// TIA Portal project "HandlingDevice" (V13)

(* hardware
DEVICE "S7300/ET200M-Station_1"  S7-300 station
   slot 0: "Profilschiene_0"  Rail  6ES7 390-1***0-0AA0
   slot 1: "PS 307 2A_1"  PS 307 2A  6ES7 307-1BA00-0AA0
   slot 2: "PLC_1"  CPU 314C-2 PN/DP  6ES7 314-6EH04-0AB0  V3.3
      slot 2: "PROFINET-Schnittstelle_1"  PN-IO
         slot 1: "Port_1"  Port
         slot 2: "Port_2"  Port
      slot 5: "DI 24/DO 16_1"  DI24/DO16
      slot 6: "AI 5/AO 2_1"  AI5/AO2
      slot 7: "Zählen_1"  Counter
      slot 8: "Positionieren_1"  Positioning
*)

// ===== PLC "PLC_1"  CPU 314C-2 PN/DP =====

VAR_GLOBAL   // PLC tag table "Standard-Variablentabelle"
   "1S1" AT %I124.0 : Bool;   // Start-Taster (NO)
   "2S1" AT %E124.1 : Bool;   // Halt-Taster (NC)
   "3S1" AT %E124.2 : Bool;   // Richten-Taster (NO)
   "1B1" AT %E124.3 : Bool;   // Zylinder A eingefahren
   "1B2" AT %E124.4 : Bool;   // Zylinder A ausgefahren
   "2B1" AT %E124.5 : Bool;   // Zylinder C in Position unten (eingefahren)
   "2B2" AT %E124.6 : Bool;   // Zylinder C in Position Werkstückaufnahme/-übergabe
   "3B1" AT %E124.7 : Bool;   // Drehtisch D in Position Werkstückaufnahme
   "3B2" AT %E125.0 : Bool;   // Drehtisch D in Position Werkstückübergabe
   "4B1" AT %E125.1 : Bool;   // Schlitten E in Position oben
   "4B2" AT %E125.2 : Bool;   // Schlitten E in Position Werkstückaufnahme/-übergabe
   "5B1" AT %E125.3 : Bool;   // Drehantrieb F in Position Werkstückaufnahme
   "5B2" AT %E125.4 : Bool;   // Drehantrieb F in Position Werkstückübergabe
   "6B1" AT %E125.5 : Bool;   // Werkstück am Greifer A angesaugt
   "6B2" AT %E125.6 : Bool;   // Werkstück am Greifer F angesaugt
   "1M1" AT %A124.0 : Bool;   // Zylinder A ausfahren
   "2M1" AT %A124.1 : Bool;   // Drehantrieb A in Position Werkstückaufnahme drehen
   "2M2" AT %A124.2 : Bool;   // Drehantrieb A in Position Werkstückübergabe drehen
   "3M1" AT %A124.3 : Bool;   // Zylinder C in Position Werkstückaufnahme/-übergabe
   "4M1" AT %A124.4 : Bool;   // Drehtisch D in Position Werkstückübergabe drehen
   "4M2" AT %A124.5 : Bool;   // Drehtisch D in Position Werkstückaufnahme drehen
   "5M1" AT %A124.6 : Bool;   // Schlitten E in Position Werkstückaufnahme/-übergabe fahren
   "6M1" AT %A124.7 : Bool;   // Drehantrieb F in Position Werkstückübergabe drehen
   "6M2" AT %A125.0 : Bool;   // Drehantrieb F in Position Werkstückaufnahme drehen
   "7M1" AT %A125.1 : Bool;   // Vakuum Greifer A einschalten
   "7M2" AT %A125.2 : Bool;   // Vakuum Greifer A ausschalten
   "8M1" AT %A125.3 : Bool;   // Vakuum Greifer F einschalten
   "8M2" AT %A125.4 : Bool;   // Vakuum Greifer F ausschalten
   "P_S" AT %A125.5 : Bool;   // Startlampe (grün)
   "P_H" AT %A125.6 : Bool;   // Haltlampe (rot)
   "P_R" AT %A125.7 : Bool;   // Richtenlampe (orange)
   "Step0" AT %M0.0 : Bool;   // Step0
   "Step1" AT %M0.1 : Bool;   // Step1
   "Step2" AT %M0.2 : Bool;   // Step2
   "Step3" AT %M0.3 : Bool;   // Step3
   "Step4" AT %M0.4 : Bool;   // Step4
   "Step5" AT %M0.5 : Bool;   // Step5
   "Step5.1" AT %M10.0 : Bool;   // Step5.1
   "Step5.2" AT %M10.1 : Bool;   // Step5.2
   "Step5.3" AT %M10.2 : Bool;   // Step5.3
   "Step5.4" AT %M10.3 : Bool;   // Step5.4
   "Step5.5" AT %M10.4 : Bool;   // Step5.5
   "Step5.6" AT %M10.5 : Bool;   // Step5.6
   "Step5.7" AT %M10.6 : Bool;   // Step5.7
   "Step5.8" AT %M10.7 : Bool;   // Step5.8
   "Step5.9" AT %M11.0 : Bool;   // Step5.9
   "Step5.10" AT %M11.1 : Bool;   // Step5.10
   "Step5.11" AT %M11.2 : Bool;   // Step5.11
   "Step5.12" AT %M11.3 : Bool;   // Step5.12
   "Step5.13" AT %M11.4 : Bool;   // Step5.13
   "Step5.14" AT %M11.5 : Bool;   // Step5.14
   "Step5.15" AT %M11.6 : Bool;   // Step5.15
   "Step5.16" AT %M11.7 : Bool;   // Step5.16
   "Step5.17" AT %M12.0 : Bool;   // Step5.17
   "InitialStep" AT %M20.0 : Bool;   // Intiral Step
   "Mx_Gerichtet" AT %M1.0 : Bool;   // Anlage Gerichtet
   "Mx_Ausgangstellung" AT %M1.1 : Bool;   // Anlage in Ausgangstellung
   "Mx_Start" AT %M1.2 : Bool;
   "Tag_1" AT %MW0 : Int;
   "Tag_2" AT %MD10 : DWord;
   "Tag_3" AT %M1.3 : Bool;
   "Tag_4" AT %QW124 : Word;
   "Tag_5" AT %M1.4 : Bool;
END_VAR

FUNCTION "FC1 Grafcet G1" : Void   // FC1, FBD
{ S7_Optimized_Access := 'FALSE' }
VERSION : 0.1
BEGIN

REGION Network 1: Step0
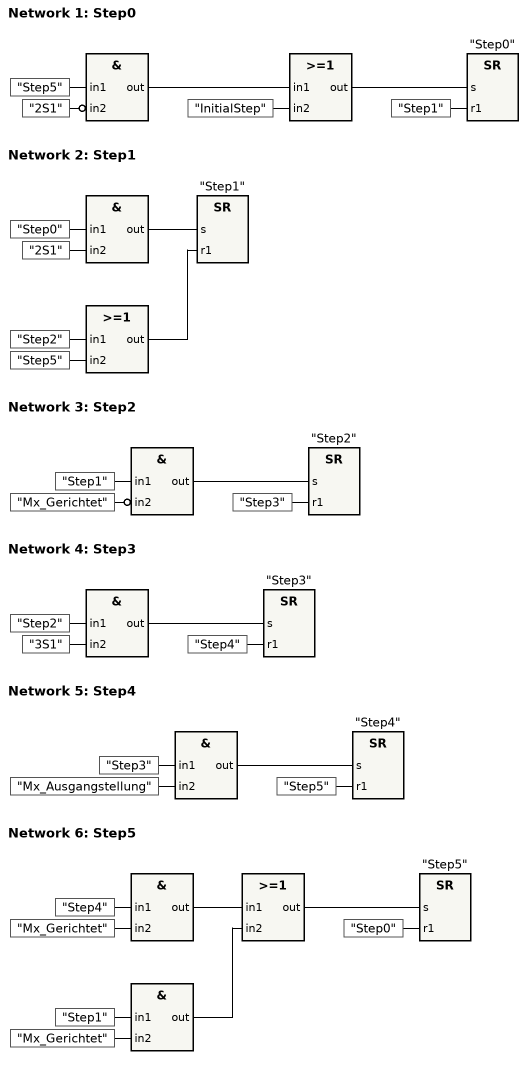
   IF ("Step5" AND NOT "2S1") OR "InitialStep" THEN
       "Step0" := TRUE;   // SR flip-flop
   END_IF;
   IF "Step1" THEN "Step0" := FALSE; END_IF;
END_REGION

REGION Network 2: Step1
   IF "Step0" AND "2S1" THEN
       "Step1" := TRUE;   // SR flip-flop
   END_IF;
   IF "Step2" OR "Step5" THEN "Step1" := FALSE; END_IF;
END_REGION

REGION Network 3: Step2
   IF "Step1" AND NOT "Mx_Gerichtet" THEN
       "Step2" := TRUE;   // SR flip-flop
   END_IF;
   IF "Step3" THEN "Step2" := FALSE; END_IF;
END_REGION

REGION Network 4: Step3
   IF "Step2" AND "3S1" THEN
       "Step3" := TRUE;   // SR flip-flop
   END_IF;
   IF "Step4" THEN "Step3" := FALSE; END_IF;
END_REGION

REGION Network 5: Step4
   IF "Step3" AND "Mx_Ausgangstellung" THEN
       "Step4" := TRUE;   // SR flip-flop
   END_IF;
   IF "Step5" THEN "Step4" := FALSE; END_IF;
END_REGION

REGION Network 6: Step5
   IF ("Step4" AND "Mx_Gerichtet") OR ("Step1" AND "Mx_Gerichtet") THEN
       "Step5" := TRUE;   // SR flip-flop
   END_IF;
   IF "Step0" THEN "Step5" := FALSE; END_IF;
END_REGION
END_FUNCTION

FUNCTION "FC2 Grafcet G5" : Void   // FC2, FBD
{ S7_Optimized_Access := 'FALSE' }
VERSION : 0.1
   VAR_TEMP   // added for the SCL form of the ladder/FBD networks
      _w1 : Bool;
   END_VAR
BEGIN

REGION Network 1: Step 5.1
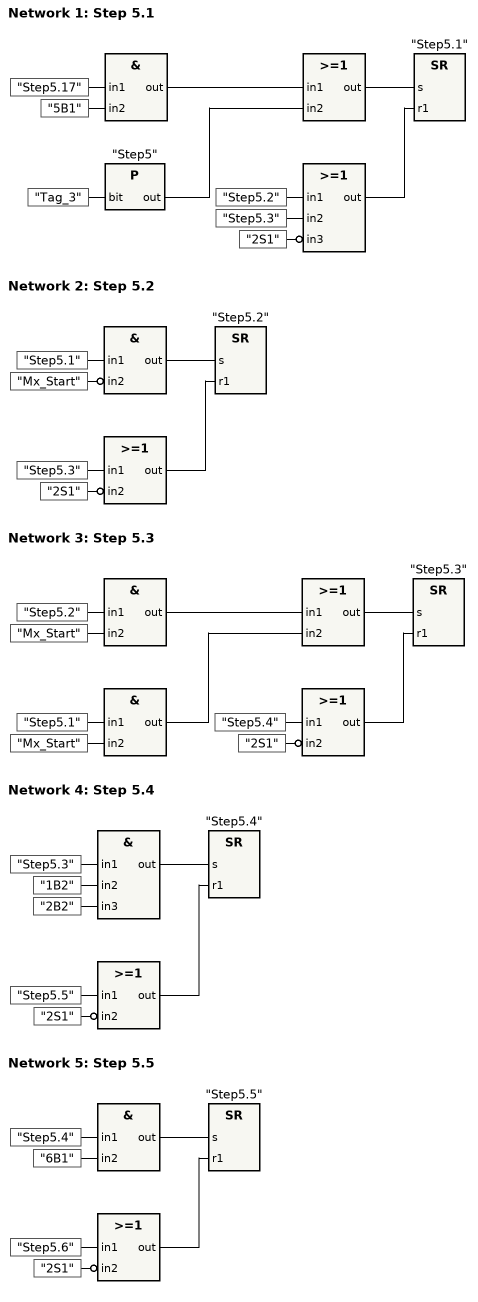
   #_w1 := "Step5" AND NOT "Tag_3";   // rising edge of "Step5"
   "Tag_3" := "Step5";
   IF ("Step5.17" AND "5B1") OR #_w1 THEN
       "Step5.1" := TRUE;   // SR flip-flop
   END_IF;
   IF "Step5.2" OR "Step5.3" OR NOT "2S1" THEN "Step5.1" := FALSE; END_IF;
END_REGION

REGION Network 2: Step 5.2
   IF "Step5.1" AND NOT "Mx_Start" THEN
       "Step5.2" := TRUE;   // SR flip-flop
   END_IF;
   IF "Step5.3" OR NOT "2S1" THEN "Step5.2" := FALSE; END_IF;
END_REGION

REGION Network 3: Step 5.3
   IF ("Step5.2" AND "Mx_Start") OR ("Step5.1" AND "Mx_Start") THEN
       "Step5.3" := TRUE;   // SR flip-flop
   END_IF;
   IF "Step5.4" OR NOT "2S1" THEN "Step5.3" := FALSE; END_IF;
END_REGION

REGION Network 4: Step 5.4
   IF "Step5.3" AND "1B2" AND "2B2" THEN
       "Step5.4" := TRUE;   // SR flip-flop
   END_IF;
   IF "Step5.5" OR NOT "2S1" THEN "Step5.4" := FALSE; END_IF;
END_REGION

REGION Network 5: Step 5.5
   IF "Step5.4" AND "6B1" THEN
       "Step5.5" := TRUE;   // SR flip-flop
   END_IF;
   IF "Step5.6" OR NOT "2S1" THEN "Step5.5" := FALSE; END_IF;
END_REGION

REGION Network 6: Step 5.6
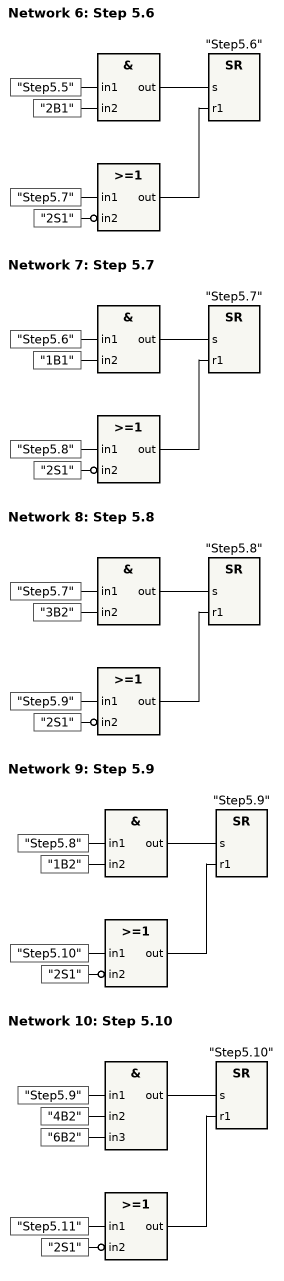
   IF "Step5.5" AND "2B1" THEN
       "Step5.6" := TRUE;   // SR flip-flop
   END_IF;
   IF "Step5.7" OR NOT "2S1" THEN "Step5.6" := FALSE; END_IF;
END_REGION

REGION Network 7: Step 5.7
   IF "Step5.6" AND "1B1" THEN
       "Step5.7" := TRUE;   // SR flip-flop
   END_IF;
   IF "Step5.8" OR NOT "2S1" THEN "Step5.7" := FALSE; END_IF;
END_REGION

REGION Network 8: Step 5.8
   IF "Step5.7" AND "3B2" THEN
       "Step5.8" := TRUE;   // SR flip-flop
   END_IF;
   IF "Step5.9" OR NOT "2S1" THEN "Step5.8" := FALSE; END_IF;
END_REGION

REGION Network 9: Step 5.9
   IF "Step5.8" AND "1B2" THEN
       "Step5.9" := TRUE;   // SR flip-flop
   END_IF;
   IF "Step5.10" OR NOT "2S1" THEN "Step5.9" := FALSE; END_IF;
END_REGION

REGION Network 10: Step 5.10
   IF "Step5.9" AND "4B2" AND "6B2" THEN
       "Step5.10" := TRUE;   // SR flip-flop
   END_IF;
   IF "Step5.11" OR NOT "2S1" THEN "Step5.10" := FALSE; END_IF;
END_REGION

REGION Network 11: Step 5.11
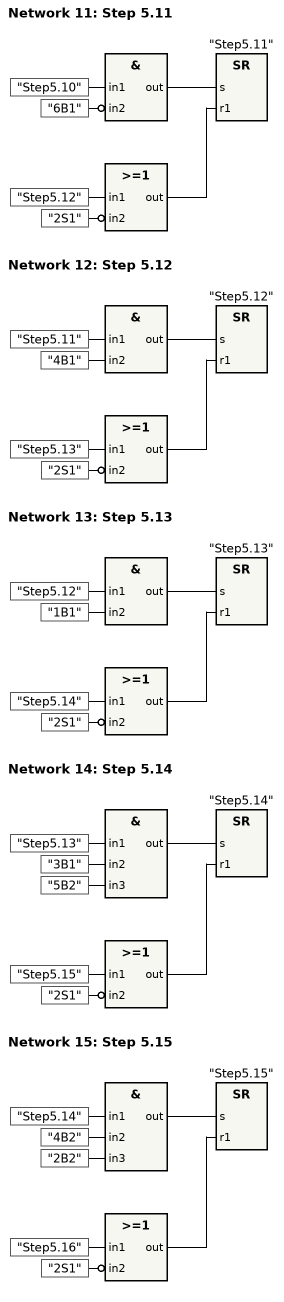
   IF "Step5.10" AND NOT "6B1" THEN
       "Step5.11" := TRUE;   // SR flip-flop
   END_IF;
   IF "Step5.12" OR NOT "2S1" THEN "Step5.11" := FALSE; END_IF;
END_REGION

REGION Network 12: Step 5.12
   IF "Step5.11" AND "4B1" THEN
       "Step5.12" := TRUE;   // SR flip-flop
   END_IF;
   IF "Step5.13" OR NOT "2S1" THEN "Step5.12" := FALSE; END_IF;
END_REGION

REGION Network 13: Step 5.13
   IF "Step5.12" AND "1B1" THEN
       "Step5.13" := TRUE;   // SR flip-flop
   END_IF;
   IF "Step5.14" OR NOT "2S1" THEN "Step5.13" := FALSE; END_IF;
END_REGION

REGION Network 14: Step 5.14
   IF "Step5.13" AND "3B1" AND "5B2" THEN
       "Step5.14" := TRUE;   // SR flip-flop
   END_IF;
   IF "Step5.15" OR NOT "2S1" THEN "Step5.14" := FALSE; END_IF;
END_REGION

REGION Network 15: Step 5.15
   IF "Step5.14" AND "4B2" AND "2B2" THEN
       "Step5.15" := TRUE;   // SR flip-flop
   END_IF;
   IF "Step5.16" OR NOT "2S1" THEN "Step5.15" := FALSE; END_IF;
END_REGION

REGION Network 16: Step 5.16
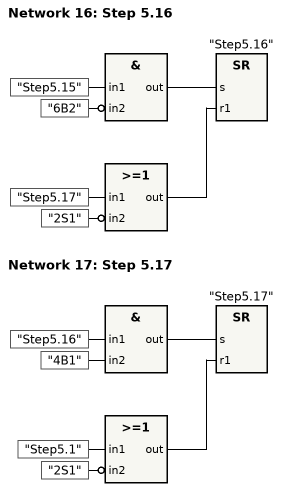
   IF "Step5.15" AND NOT "6B2" THEN
       "Step5.16" := TRUE;   // SR flip-flop
   END_IF;
   IF "Step5.17" OR NOT "2S1" THEN "Step5.16" := FALSE; END_IF;
END_REGION

REGION Network 17: Step 5.17
   IF "Step5.16" AND "4B1" THEN
       "Step5.17" := TRUE;   // SR flip-flop
   END_IF;
   IF "Step5.1" OR NOT "2S1" THEN "Step5.17" := FALSE; END_IF;
END_REGION
END_FUNCTION

FUNCTION "FC3 Action" : Void   // FC3, FBD
{ S7_Optimized_Access := 'FALSE' }
VERSION : 0.1
BEGIN

REGION Network 1: Richtenlampe (orange)
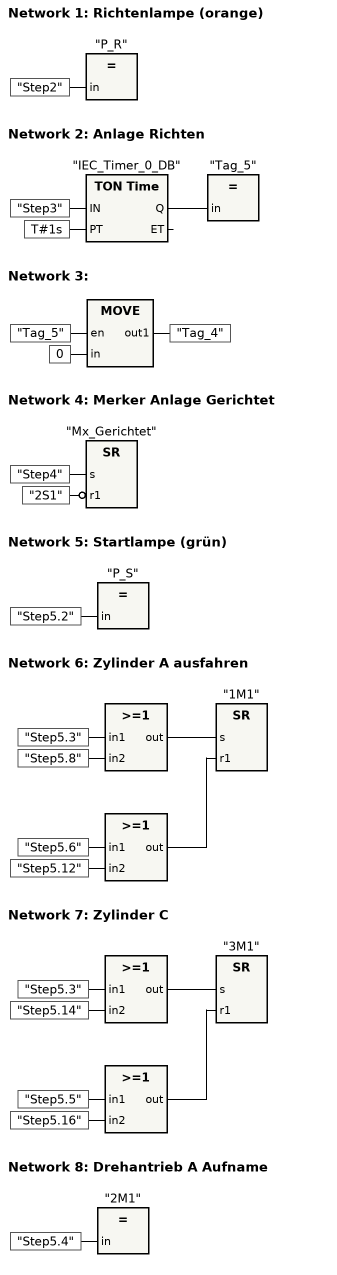
   "P_R" := "Step2";
END_REGION

REGION Network 2: Anlage Richten
   "IEC_Timer_0_DB".TON(IN := "Step3", PT := T#1s);
   "Tag_5" := "IEC_Timer_0_DB".Q;
END_REGION

REGION Network 3
   IF "Tag_5" THEN "Tag_4" := 0; END_IF;
END_REGION

REGION Network 4: Merker Anlage Gerichtet
   IF "Step4" THEN
       "Mx_Gerichtet" := TRUE;   // SR flip-flop
   END_IF;
   IF NOT "2S1" THEN "Mx_Gerichtet" := FALSE; END_IF;
END_REGION

REGION Network 5: Startlampe (grün)
   "P_S" := "Step5.2";
END_REGION

REGION Network 6: Zylinder A ausfahren
   IF "Step5.3" OR "Step5.8" THEN
       "1M1" := TRUE;   // SR flip-flop
   END_IF;
   IF "Step5.6" OR "Step5.12" THEN "1M1" := FALSE; END_IF;
END_REGION

REGION Network 7: Zylinder C
   IF "Step5.3" OR "Step5.14" THEN
       "3M1" := TRUE;   // SR flip-flop
   END_IF;
   IF "Step5.5" OR "Step5.16" THEN "3M1" := FALSE; END_IF;
END_REGION

REGION Network 8: Drehantrieb A Aufname
   "2M1" := "Step5.4";
END_REGION

REGION Network 9: Drehantribe A Abgabe
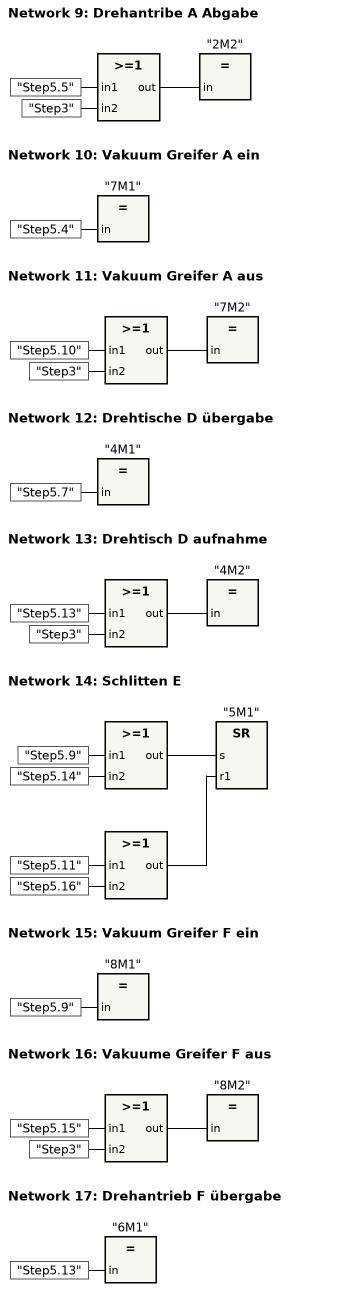
   "2M2" := "Step5.5" OR "Step3";
END_REGION

REGION Network 10: Vakuum Greifer A ein
   "7M1" := "Step5.4";
END_REGION

REGION Network 11: Vakuum Greifer A aus
   "7M2" := "Step5.10" OR "Step3";
END_REGION

REGION Network 12: Drehtische D übergabe
   "4M1" := "Step5.7";
END_REGION

REGION Network 13: Drehtisch D aufnahme
   "4M2" := "Step5.13" OR "Step3";
END_REGION

REGION Network 14: Schlitten E
   IF "Step5.9" OR "Step5.14" THEN
       "5M1" := TRUE;   // SR flip-flop
   END_IF;
   IF "Step5.11" OR "Step5.16" THEN "5M1" := FALSE; END_IF;
END_REGION

REGION Network 15: Vakuum Greifer F ein
   "8M1" := "Step5.9";
END_REGION

REGION Network 16: Vakuume Greifer F aus
   "8M2" := "Step5.15" OR "Step3";
END_REGION

REGION Network 17: Drehantrieb F übergabe
   "6M1" := "Step5.13";
END_REGION

REGION Network 18: Drehantreib F aufnahme
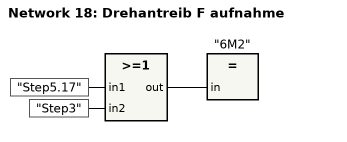
   "6M2" := "Step5.17" OR "Step3";
END_REGION
END_FUNCTION

ORGANIZATION_BLOCK "Main"   // OB1, FBD
TITLE = "Main Program Sweep (Cycle)"
{ S7_Optimized_Access := 'FALSE' }
VERSION : 0.1
BEGIN

REGION Network 1
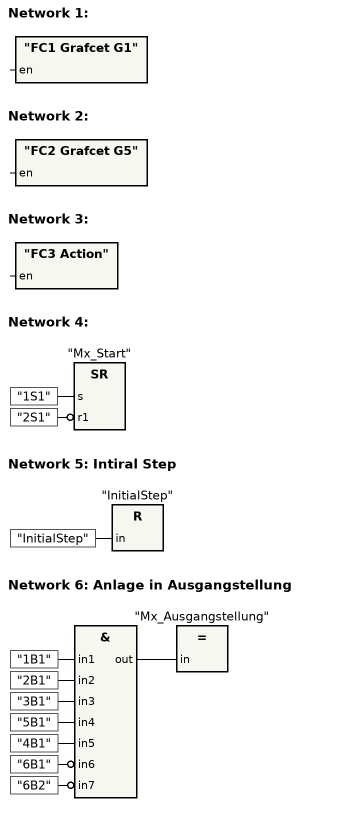
   "FC1 Grafcet G1"();
END_REGION

REGION Network 2
   "FC2 Grafcet G5"();
END_REGION

REGION Network 3
   "FC3 Action"();
END_REGION

REGION Network 4
   IF "1S1" THEN
       "Mx_Start" := TRUE;   // SR flip-flop
   END_IF;
   IF NOT "2S1" THEN "Mx_Start" := FALSE; END_IF;
END_REGION

REGION Network 5: Intiral Step
   IF "InitialStep" THEN "InitialStep" := FALSE; END_IF;
END_REGION

REGION Network 6: Anlage in Ausgangstellung
   "Mx_Ausgangstellung" := "1B1" AND "2B1" AND "3B1" AND "5B1" AND "4B1" AND NOT "6B1" AND NOT "6B2";
END_REGION
END_ORGANIZATION_BLOCK

ORGANIZATION_BLOCK "COMPLETE RESTART"   // OB100, FBD
TITLE = "Complete Restart"
{ S7_Optimized_Access := 'FALSE' }
VERSION : 0.1
BEGIN

REGION Network 1: Intiral Step
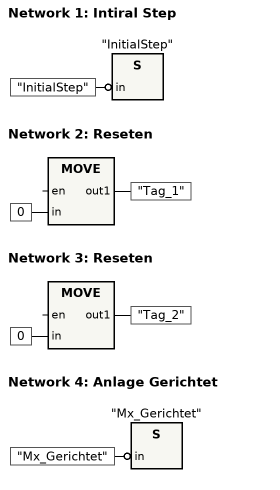
   IF NOT "InitialStep" THEN "InitialStep" := TRUE; END_IF;
END_REGION

REGION Network 2: Reseten
   "Tag_1" := 0;
END_REGION

REGION Network 3: Reseten
   "Tag_2" := 0;
END_REGION

REGION Network 4: Anlage Gerichtet
   IF NOT "Mx_Gerichtet" THEN "Mx_Gerichtet" := TRUE; END_IF;
END_REGION
END_ORGANIZATION_BLOCK